(* IEC 61131-3 sources: s22-soft-shell/ST_resources/ST programs for testing/unimplemented/parsing, 7 files *)

(* ---- CounterInOutFunction.st ---- *)
// This function is designed to test IN_OUT variable.
// Takes in_out integer and adds 1 to it "counting up by 1"
// Then returns new count with variable instead of by function name
// function name returns true to indicate success
FUNCTION CounterInOutFunction : BOOL //BOOL is the return parameter data type
VAR_IN_OUT
  InOut1 :	INT; //IN_OUT parameter
END_VAR

  InOut1 := InOut1 + 1;

  CounterFunction:= 'TRUE'; //Set the return parameter

END_FUNCTION

(* ---- CounterOutputFunction.st ---- *)
// This function is designed to test Output variable.
// Takes input integer and adds 1 to it "counting up by 1"
// Then returns new count using Output variable instead of function name
// function name returns true to indicate success
FUNCTION CounterOutputFunction : BOOL //BOOL is the return parameter data type
VAR_INPUT
  Input1 :	INT; //Input parameter
END_VAR
VAR_OUTPUT
  Output1 :	INT; //Output parameter
END_VAR

  Output1 := Input1 + 1;

  CounterFunction:= 'TRUE'; //Set the return parameter

END_FUNCTION

(* ---- ThreeVarFunction.st ---- *)
// This function is designed to test Output variable.
// Takes input integer and adds 1 to it "counting up by 1"
// Then returns new count using Output variable instead of function name
// function name returns true to indicate success
FUNCTION ThreeVarFunction : BOOL //BOOL is the return parameter data type
VAR_INPUT
  Input1 :	INT; //Input parameter
END_VAR
VAR_OUTPUT
  Output1 :	INT; //Output parameter
END_VAR
VAR_OUTPUT
  InOut1 :	INT; //Output parameter
END_VAR

  Output1 := Input1 + 1;

  InOut1  := InOut1 + 2;

  CounterFunction:= 'TRUE'; //Set the return parameter

END_FUNCTION

(* ---- 09_Main_Counter_InOut.st ---- *)
//Testing counter, increments input by one by returning value from Output variable
//
PROGRAM 09_Main_Counter_InOut
    VAR
	a : int;
        b : int;
        result0 : int;
        result1 : int;

    END_VAR
        a := 4;
        b := 2;

        // IN_OUT variable get copied into function and copied out changing the original variable when done
        result0 := CounterInOutFunction(InOut1 := a); // expects result of true and a as 5

        result1 := CounterInOutFunction(InOut1 := b); // expects result of true and b as 3

END_PROGRAM

(* ---- 09_Main_Counter_Output.st ---- *)
//Testing counter, increments input by one by returning value from Output variable
PROGRAM 09_Main_Counter_Output
    VAR
	a : int;
        b : int;
        result0 : int;
        result1 : int;

    END_VAR
        a := 0;
        b := 0;

        // Output variables in a function call use => instead of := because Output variable is not being
        // assinged an initial value but rather it will only be outputing a value to that variable.
        result0 := CounterOutputFunction( Input1 := 4, Output1 => a); // expects result of true and a as 5

        result1 := CounterOutputFunction(Input1 := 2, Output1 => b); // expects result of true and b as 3

END_PROGRAM

(* ---- 09_Main_Demo_01.st ---- *)
// Testing for GO West Example use case example
// program doesnt go into while loop without C API
// is used to set INPUT1 or INPUT2 to TRUE
// x represents number of loops INPUT1 and INPUT2 are both true during
// OUTPUT1 represents number of loops
PROGRAM 09_Main_Demo_01
    VAR
	x : int;
        INPUT1 : bool;
        INPUT2 : bool;
        OUTPUT1 : int;
    END_VAR
        x := 0;
        INPUT1 := False;
        INPUT2 := False ;
        OUTPUT1 : 0;
//API would control INPUTs after here HERE here

        WHILE (INPUT1) OR (INPUT2) DO
            If (INPUT1) AND (INPUT2) THEN
                x:= x +1
            END_IF;
            OUTPUT1 := SimpleAddFunction(Input1 := OUTPUT1, Input2 := 1);
        END_WHILE;

END_PROGRAM

(* ---- 09_Main_ThreeVar.st ---- *)
//Testing for INPUT, OUTPUT, IN_OUT type variables in same function call
PROGRAM 09_Main_ThreeVar
    VAR
	a : int;
        b : int;
        result0 : int;
    END_VAR
        a := 0;
        b := 0;

        // Output variables in a function call use => instead of := because Output variable is not being
        // assinged an initial value but rather it will only be outputing a value to that variable.
        // expects result of true, a as 5 and b as 2
        result0 := CounterOutputFunction( Input1 := 4, Output1 => a, InOut1 := b);

END_PROGRAM
